{attribute 'linkalways'} 
{attribute 'no_explicit_call' := 'This FB is a CLASS and must be accessed using methods or properties'}
{attribute 'enable_dynamic_creation'}
FUNCTION_BLOCK INTERNAL AsyncCommandStateMachine IMPLEMENTS AsyncCommandStateControl
VAR
	state : (IDLE, INITIALIZING, EXECUTING, COMPLETING, COMPLETED, ABORTING, ABORTED, ERRORED);
	_errorId : UDINT;
END_VAR

METHOD PUBLIC Abort
VAR_INPUT
END_VAR
CASE state OF
	IDLE : RETURN;
	ABORTING : RETURN;
	COMPLETED : RETURN;
	ABORTED : RETURN;
	ERRORED : RETURN;
END_CASE

state := ABORTING;
END_METHOD

METHOD PUBLIC Error
VAR_INPUT
	ErrorId : UDINT;
END_VAR
CASE state OF
	IDLE : RETURN;
	COMPLETED : RETURN;
	ABORTED : RETURN;
	ERRORED : RETURN;
END_CASE

_errorId := ErrorId;
state := ERRORED;
END_METHOD

{attribute 'monitoring' := 'call'}
PROPERTY PUBLIC ErrorId : UDINT
GET
ErrorID := _errorId;
END_GET
END_PROPERTY

METHOD PUBLIC Execute
VAR_INPUT
END_VAR
CASE state OF
	INITIALIZING : RETURN;
	EXECUTING : RETURN;
	COMPLETING : RETURN;
	ABORTING : RETURN;
END_CASE

_errorId := 0;
state := INITIALIZING;
END_METHOD

{attribute 'monitoring' := 'call'}
PROPERTY PUBLIC IsAborted : BOOL
GET
IsAborted := state = ABORTED;
END_GET
END_PROPERTY

{attribute 'monitoring' := 'call'}
PROPERTY PUBLIC IsAborting : BOOL
GET
IsAborting := state = ABORTING;
END_GET
END_PROPERTY

{attribute 'monitoring' := 'call'}
PROPERTY PUBLIC IsCompleted : BOOL
GET
IsCompleted := state = COMPLETED;
END_GET
END_PROPERTY

{attribute 'monitoring' := 'call'}
PROPERTY PUBLIC IsCompleting : BOOL
GET
IsCompleting := state = COMPLETING;
END_GET
END_PROPERTY

{attribute 'monitoring' := 'call'}
PROPERTY PUBLIC IsErrored : BOOL
GET
IsErrored := state = ERRORED;
END_GET
END_PROPERTY

{attribute 'monitoring' := 'call'}
PROPERTY PUBLIC IsExecuting : BOOL
GET
IsExecuting := state = EXECUTING;
END_GET
END_PROPERTY

{attribute 'monitoring' := 'call'}
PROPERTY PUBLIC IsIdle : BOOL
GET
IsIdle:= state = IDLE;
END_GET
END_PROPERTY

{attribute 'monitoring' := 'call'}
PROPERTY PUBLIC IsInitializing : BOOL
GET
IsInitializing := state = INITIALIZING;
END_GET
END_PROPERTY

METHOD PUBLIC Next
VAR_INPUT
END_VAR
CASE state OF
	IDLE : RETURN;
	INITIALIZING : StateComplete_Initializing();
	EXECUTING : StateComplete_Executing();
	COMPLETING : StateComplete_Completing();
	COMPLETED : RETURN;
	ABORTING : StateComplete_Aborting();
	ABORTED : RETURN;
	ERRORED : RETURN;
END_CASE
END_METHOD

METHOD PRIVATE StateComplete_Aborting
VAR_INPUT
END_VAR
state := ABORTED;
END_METHOD

METHOD PRIVATE StateComplete_Completing
VAR_INPUT
END_VAR
state := COMPLETED;
END_METHOD

METHOD PRIVATE StateComplete_Executing
VAR_INPUT
END_VAR
state := COMPLETING;
END_METHOD

METHOD PRIVATE StateComplete_Initializing
VAR_INPUT
END_VAR
state := EXECUTING;
END_METHOD

END_FUNCTION_BLOCK

(* stored: Version 1.1.0.1
   POU AsyncCommandStateMachine: Id {0c151bef-3f58-41ba-87ee-1d343a471019}, SpecialFunc None
   Folder Private: Id {9e4bb0f2-8bca-02be-22c5-c88b3f4896ba}
   Method Abort: Id {a7cbfa36-7269-07ed-3a90-212389d128d9}
   Method Error: Id {c7df7efb-bf18-08a9-0a54-f9e36845dc8f}
   Property ErrorId: Id {1ae5ea41-9381-0ea0-1e7d-e01c680093ef}
   Get Get: Id {177e6653-5236-0183-0d8d-5297a1a36010}
   Method Execute: Id {636f1081-2a8a-0d25-0e8c-4df17c4a8ab0}
   Property IsAborted: Id {463c2c3e-b1e3-03c8-2463-a42d3ac062e2}
   Get Get: Id {d423c7da-cedb-0ed8-150c-780c4a9546db}
   Property IsAborting: Id {dbb94993-6904-0ff3-3e11-e586757361e1}
   Get Get: Id {4f562a40-dbb9-010a-35d7-88202a14b292}
   Property IsCompleted: Id {bdf352ba-8f2e-0342-1514-ad3b845a8d2e}
   Get Get: Id {da04174c-7b98-018d-25cb-bc9c812ef9d5}
   Property IsCompleting: Id {206fc9ca-6d74-0427-3db4-63aa13e11585}
   Get Get: Id {aa9b89c5-d895-0667-1418-5d5779238f1c}
   Property IsErrored: Id {209a7060-c21e-088d-1c58-dacb5ee3abca}
   Get Get: Id {b4e7aff5-59d2-0e97-3e8b-1aec9212179b}
   Property IsExecuting: Id {e9ca9061-6d01-0b57-39c9-49918756cbdc}
   Get Get: Id {309c7707-65bc-06eb-0844-8020e54f8f5a}
   Property IsIdle: Id {8d51b4cb-8025-0ea9-071e-08691b1fe6d6}
   Get Get: Id {531d2b82-b858-0a02-0cdd-6d9e42212b53}
   Property IsInitializing: Id {46d4bbef-6352-0501-3e35-41623a34642a}
   Get Get: Id {1e6ff335-6789-0891-2a6b-ce3b8cc53654}
   Method Next: Id {0bcee425-e887-0a4c-3a01-fa64bbb61979}
   Method StateComplete_Aborting: Id {8d511f27-c5a2-03dd-263d-b902dac1e354}
   Method StateComplete_Completing: Id {99e185bf-d474-001a-13ad-ee4d830f6985}
   Method StateComplete_Executing: Id {cecb7746-f794-07fe-391e-f9bec990ec21}
   Method StateComplete_Initializing: Id {4e1ba278-4215-0723-25c1-681afe132e99} *)
